FUNCTION F_EventTimeStamp
VAR_IN_OUT
	stEvent : ST_Event;
END_VAR
VAR
	stFileTime : T_FILETIME;
	fbGetSystemTime : GETSYSTEMTIME;
END_VAR

fbGetSystemTime(timeLoDW => stFileTime.dwLowDateTime, timeHiDW => stfiletime.dwHighDateTime);
stEvent.tTimeStamp := FileTime_To_Dt(filetime := stFileTime);

END_FUNCTION

(* stored: Version 1.1.0.1, ProductVersion 3.1.4024.9
   POU F_EventTimeStamp: Id {803a4ffa-4675-47f5-bef6-21aa213b69b6}, SpecialFunc None *)
